PROGRAM StartStop
VAR
	StartPb			:	BOOL;	// start switch (NO)
	StopPb			:	BOOL;	// stop switch (NC)
	Motor1			:	BOOL;	// run conveyor 1 belt
	Motor2			:	BOOL;	// run conveyor 2 belt	
END_VAR
VAR // added by the converter: edge detectors and wires of the graphical bodies
    _w1 : BOOL;
END_VAR

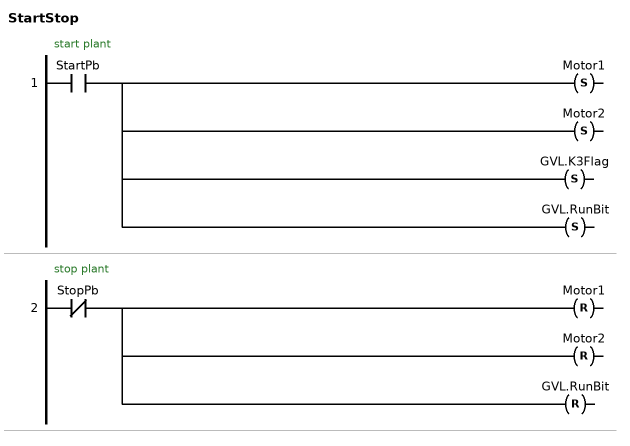
// NETWORK 1
// start plant
Motor1 S= StartPb;
Motor2 S= StartPb;
GVL.K3Flag S= StartPb;
GVL.RunBit S= StartPb;

// NETWORK 2
// stop plant
_w1 := NOT StopPb;
Motor1 R= _w1;
Motor2 R= _w1;
GVL.RunBit R= _w1;

END_PROGRAM

(* stored: Version 1.1.0.1, ProductVersion 3.1.4024.15
   POU StartStop: Id {16b51bd3-7f43-4cc4-aaf2-52d03ab3042f}, SpecialFunc None *)
